(* IEC 61131-3 sources: Eaton-PLC-CSV-MQTT/CSV-MQTT/scripts/Functions, 4 files *)

(* ---- F_AssignField.st ---- *)
// Helper function to assign a string value to a specific field in ST_CSVRow
// Uses pointer manipulation to access structure fields dynamically
FUNCTION F_AssignField : BOOL
VAR_INPUT
    pStruct    : POINTER TO ST_CSVRow;  // Pointer to the CSV row structure
    iFieldNum  : INT;                   // Field number (1-13)
    sValue     : STRING(64);            // Value to assign
END_VAR

// Validate inputs
IF pStruct = 0 OR iFieldNum < 1 OR iFieldNum > 13 THEN
    F_AssignField := FALSE;
    RETURN;
END_IF;

// Assign value to appropriate field based on field number
CASE iFieldNum OF
    1:  pStruct^.Col1  := sValue;
    2:  pStruct^.Col2  := sValue;
    3:  pStruct^.Col3  := sValue;
    4:  pStruct^.Col4  := sValue;
    5:  pStruct^.Col5  := sValue;
    6:  pStruct^.Col6  := sValue;
    7:  pStruct^.Col7  := sValue;
    8:  pStruct^.Col8  := sValue;
    9:  pStruct^.Col9  := sValue;
    10: pStruct^.Col10 := sValue;
    11: pStruct^.Col11 := sValue;
    12: pStruct^.Col12 := sValue;
    13: pStruct^.Col13 := sValue;
END_CASE;

F_AssignField := TRUE;

(* ---- F_BuildJsonFromRow.st ---- *)
// Helper function to build JSON string from CSV row structure
// Formats data as: {"Col1":"value1","Col2":"value2",...}
FUNCTION F_BuildJsonFromRow : BOOL
VAR_INPUT
    row : ST_CSVRow;           // Input CSV row data
END_VAR
VAR_IN_OUT
    sJson : STRING(2048);      // Output JSON string
END_VAR

// Build JSON manually since library functions may vary
sJson := '{';

// Add each column as a JSON key-value pair
sJson := CONCAT(sJson, '"Col1":"');  sJson := CONCAT(sJson, row.Col1);  sJson := CONCAT(sJson, '",');
sJson := CONCAT(sJson, '"Col2":"');  sJson := CONCAT(sJson, row.Col2);  sJson := CONCAT(sJson, '",');
sJson := CONCAT(sJson, '"Col3":"');  sJson := CONCAT(sJson, row.Col3);  sJson := CONCAT(sJson, '",');
sJson := CONCAT(sJson, '"Col4":"');  sJson := CONCAT(sJson, row.Col4);  sJson := CONCAT(sJson, '",');
sJson := CONCAT(sJson, '"Col5":"');  sJson := CONCAT(sJson, row.Col5);  sJson := CONCAT(sJson, '",');
sJson := CONCAT(sJson, '"Col6":"');  sJson := CONCAT(sJson, row.Col6);  sJson := CONCAT(sJson, '",');
sJson := CONCAT(sJson, '"Col7":"');  sJson := CONCAT(sJson, row.Col7);  sJson := CONCAT(sJson, '",');
sJson := CONCAT(sJson, '"Col8":"');  sJson := CONCAT(sJson, row.Col8);  sJson := CONCAT(sJson, '",');
sJson := CONCAT(sJson, '"Col9":"');  sJson := CONCAT(sJson, row.Col9);  sJson := CONCAT(sJson, '",');
sJson := CONCAT(sJson, '"Col10":"'); sJson := CONCAT(sJson, row.Col10); sJson := CONCAT(sJson, '",');
sJson := CONCAT(sJson, '"Col11":"'); sJson := CONCAT(sJson, row.Col11); sJson := CONCAT(sJson, '",');
sJson := CONCAT(sJson, '"Col12":"'); sJson := CONCAT(sJson, row.Col12); sJson := CONCAT(sJson, '",');
sJson := CONCAT(sJson, '"Col13":"'); sJson := CONCAT(sJson, row.Col13); sJson := CONCAT(sJson, '"');

sJson := CONCAT(sJson, '}');

F_BuildJsonFromRow := TRUE;

(* ---- F_GetNextLine.st ---- *)
// Helper function to extract next line from a string buffer
// Returns TRUE if a line was found, FALSE if end of buffer reached
FUNCTION F_GetNextLine : BOOL
VAR_INPUT
    sBuffer    : STRING(4096);  // Input buffer containing multiple lines
    iStartPos  : INT;           // Starting position to search from
END_VAR
VAR_OUTPUT
    sLine      : STRING(512);   // Extracted line (without line break)
    iEndPos    : INT;           // Position after the line break
END_VAR
VAR
    i          : INT;
    iLen       : INT;
    iLineLen   : INT := 0;
    cChar      : BYTE;
END_VAR

// Initialize
sLine := '';
iLen := LEN(sBuffer);

// Check if we're at or past end of buffer
IF iStartPos > iLen OR iStartPos < 1 THEN
    F_GetNextLine := FALSE;
    RETURN;
END_IF;

// Extract characters until newline or end of buffer
FOR i := iStartPos TO iLen DO
    cChar := sBuffer[i];

    // Check for line break characters (LF=10, CR=13)
    IF cChar = 10 OR cChar = 13 THEN
        iEndPos := i;

        // Handle CRLF (skip the LF if next char is LF)
        IF cChar = 13 AND i < iLen THEN
            IF sBuffer[i+1] = 10 THEN
                iEndPos := i + 1;
            END_IF;
        END_IF;

        F_GetNextLine := TRUE;
        RETURN;
    END_IF;

    // Append character to line
    IF iLineLen < 511 THEN
        iLineLen := iLineLen + 1;
        sLine[iLineLen] := cChar;
    END_IF;
END_FOR;

// Reached end of buffer - return last line if any content found
IF iLineLen > 0 THEN
    iEndPos := iLen;
    F_GetNextLine := TRUE;
ELSE
    F_GetNextLine := FALSE;
END_IF;

(* ---- F_ParseCSVLine.st ---- *)
// Parses a CSV line into a structured data type with 13 columns
// Splits string by semicolon delimiter and handles quoted fields
FUNCTION F_ParseCSVLine : ST_CSVRow
VAR_INPUT
    sLine : STRING(512);  // Input: CSV line (e.g., "val1;val2;val3;...")
END_VAR
VAR
    result      : ST_CSVRow;
    sField      : STRING(64);
    iPos        : INT := 1;
    iFieldNum   : INT := 0;
    iLen        : INT;
    bInQuotes   : BOOL := FALSE;
    cChar       : BYTE;
    i           : INT;
    iFieldLen   : INT := 0;
END_VAR

iLen := LEN(sLine);

// Parse through the line character by character
FOR i := 1 TO iLen DO
    cChar := sLine[i];

    // Handle quote character
    IF cChar = 34 THEN  // ASCII 34 = double quote
        bInQuotes := NOT bInQuotes;
        // Don't add quotes to field content

    // Handle semicolon delimiter (only if not inside quotes)
    ELSIF cChar = 59 AND NOT bInQuotes THEN  // ASCII 59 = semicolon
        iFieldNum := iFieldNum + 1;
        F_AssignField(ADR(result), iFieldNum, sField);
        sField := '';
        iFieldLen := 0;

    // Regular character - add to current field
    ELSE
        IF iFieldLen < 63 THEN
            iFieldLen := iFieldLen + 1;
            sField[iFieldLen] := cChar;
        END_IF;
    END_IF;
END_FOR;

// Assign last field
IF iFieldNum < 13 THEN
    iFieldNum := iFieldNum + 1;
    F_AssignField(ADR(result), iFieldNum, sField);
END_IF;

F_ParseCSVLine := result;
